(*

.. <legal notes>

legal notes
=================
| SPDX-FileCopyrightText: © 2026 Oleksandr Tiutyk <trofimich@gmail.com>
| SPDX-License-Identifier: LGPL-3.0-only
| For details check: LGPL-3.0-only_

.. _LGPL-3.0-only: https://www.gnu.org/licenses/lgpl-3.0.en.html

.. </legal notes>

*)

FUNCTION_BLOCK ABSTRACT AutomationController 
VAR_GENERIC CONSTANT
    _DeviceCount : INT(0..1000) := 0;
END_VAR
EXTENDS Automation.AutomationComponent IMPLEMENTS IAutomationController
VAR
	_ExceptionHandler : Core.IExceptionHandler;

	_State : AUTOMATION_CONTROLLER_STATE;	
	_PreviousState : AUTOMATION_CONTROLLER_STATE;	

	_Diagnostics : AUTOMATION_CONTROLLER_DIAGNOSTICS;
END_VAR

{attribute 'monitoring' := 'call'}
PROPERTY DeviceCount : INT
GET
DeviceCount := _DeviceCount;
END_GET
END_PROPERTY

{attribute 'monitoring' := 'call'}
PROPERTY ABSTRACT Devices : REFERENCE TO ARRAY [0.._DeviceCount - 1] OF Automation.IDevice
GET
END_GET
END_PROPERTY

{attribute 'monitoring' := 'call'}
PROPERTY FINAL Diagnostics : REFERENCE TO AUTOMATION_CONTROLLER_DIAGNOSTICS
GET
Diagnostics REF= _Diagnostics;
END_GET
END_PROPERTY

METHOD FINAL Disable
VAR
	i : INT;

	exceptionCode : __SYSTEM.ExceptionCode;
	exception : Core.IException;
END_VAR
__TRY
	IF _Enabled THEN
		OnEnabledChanging(FALSE);
	END_IF
	
	IF __ISVALIDREF(Devices) AND_THEN _DeviceCount > 0 THEN
		FOR i := 0 TO _DeviceCount - 1 DO
			Devices[i].Disable();
		END_FOR	
	END_IF

	IF _Enabled THEN	
		_Enabled := FALSE;
		
		OnEnabledChanged();
	END_IF
__CATCH(exceptionCode)	
	_State := AUTOMATION_CONTROLLER_STATE.FAULT;

	exception := Core.ExceptionManager.GetLastException(exceptionCode);	

	fillErrorLog('LastDisableError', Diagnostics.LastDisableError, exception);					
__ENDTRY
END_METHOD

METHOD FINAL Enable
VAR_INPUT
	includeChildren : BOOL := TRUE;
END_VAR
VAR
	i : INT;

	exceptionCode : __SYSTEM.ExceptionCode;
	exception : Core.IException;
END_VAR
__TRY
	IF NOT _Enabled THEN
		OnEnabledChanging(TRUE);
	END_IF
	
	IF includeChildren AND_THEN __ISVALIDREF(Devices) AND_THEN _DeviceCount > 0 THEN
		FOR i := 0 TO _DeviceCount - 1 DO
			Devices[i].Enable();
		END_FOR	
	END_IF
	
	IF NOT _Enabled THEN
		_Enabled := TRUE;
		
		OnEnabledChanged();
	END_IF
__CATCH(exceptionCode)	
	_State := AUTOMATION_CONTROLLER_STATE.FAULT;

	exception := Core.ExceptionManager.GetLastException(exceptionCode);	

	fillErrorLog('LastEnableError', Diagnostics.LastEnableError, exception);					
__ENDTRY
END_METHOD

PROPERTY FINAL ExceptionHandler : Core.IExceptionHandler
GET
ExceptionHandler := _ExceptionHandler;
END_GET
SET
_ExceptionHandler := ExceptionHandler;
END_SET
END_PROPERTY

METHOD FINAL Execute
VAR
	invalidStateException : Core.StandardException;
END_VAR
_PreviousState := _State;

IF NOT Enabled THEN
	RETURN;
END_IF

IF _State = AUTOMATION_CONTROLLER_STATE.INITIAL THEN
	invalidStateException.Throw(NamespaceName, ClassName, __POUNAME(), __POSITION(), "Automation controller is not initialized");
END_IF

handleInputDevices();

handleWorkingStates();

handleOutputDevices();
END_METHOD

METHOD FB_init : BOOL
VAR_INPUT
	(* if TRUE, the retain variables are initialized (warm start / cold start)*)
	bInitRetains	: BOOL;
	(* if TRUE, the instance afterwards gets moved into the copy code (online change)*)
	bInCopyCode	: BOOL;
	name : WSTRING;
END_VAR
_Name := SEL(Core.WideStrings.IsNullOrWhiteSpace(name), name, GetDefaultName());
END_METHOD

METHOD PRIVATE fillErrorLog
VAR_INPUT
	errorPlace : STRING(39);
END_VAR
VAR_IN_OUT
	targetErrorLog : AUTOMATION_ERROR_LOG;
	sourceException : Core.IException;  
END_VAR
_Diagnostics.LastErrorPalce := errorPlace;

targetErrorLog.ShortMessage := sourceException.GetMessage(FALSE, FALSE);
targetErrorLog.FullMessage := sourceException.GetMessage(TRUE, TRUE);
targetErrorLog.Source := sourceException.GetSourceDescription();
targetErrorLog.LocalTimestamp := sourceException.LocalTimestamp;
targetErrorLog.UtcTimestamp := sourceException.UtcTimestamp;

Core.LogManager.TryLogException(sourceException, "AutomationControllerError");
END_METHOD

METHOD PRIVATE handleInputDevices
VAR
	i : DINT;

	exceptionCode : __SYSTEM.ExceptionCode;
	exception : Core.IException;
	
	inputDevice : Automation.IInputDevice;
END_VAR
IF __ISVALIDREF(Devices) AND_THEN _DeviceCount > 0 THEN
	FOR i := 0 TO _DeviceCount - 1 DO
		IF NOT Devices[i].Enabled OR_ELSE NOT __QUERYINTERFACE(Devices[i], inputDevice) THEN
			CONTINUE;
		END_IF
		
		__TRY
			inputDevice.ProcessInput();
		__CATCH(exceptionCode)
			exception := Core.ExceptionManager.GetLastException(exceptionCode);
						
			fillErrorLog('LastRefreshInputDeviceError', Diagnostics.LastRefreshInputDeviceError, exception);
					
			IF _State <> AUTOMATION_CONTROLLER_STATE.FAULT THEN
				setState(AUTOMATION_CONTROLLER_STATE.FAULT);				
			END_IF					
		__ENDTRY
	END_FOR
END_IF
END_METHOD

METHOD PRIVATE handleOutputDevices
VAR
	i : DINT;

	exceptionCode : __SYSTEM.ExceptionCode;
	exception : Core.IException;
	
	outputDevice : Automation.IOutputDevice;	
END_VAR
IF __ISVALIDREF(Devices) AND_THEN _DeviceCount > 0 THEN
	FOR i := 0 TO _DeviceCount - 1 DO
		IF NOT Devices[i].Enabled OR_ELSE NOT __QUERYINTERFACE(Devices[i], outputDevice) THEN
			CONTINUE;
		END_IF
		
		__TRY
			outputDevice.ProcessOutput(); 
		__CATCH(exceptionCode)
			exception := Core.ExceptionManager.GetLastException(exceptionCode);
						
			fillErrorLog('LastRefreshOutputDeviceError', Diagnostics.LastRefreshOutputDeviceError, exception);

			IF _State <> AUTOMATION_CONTROLLER_STATE.FAULT THEN
				setState(AUTOMATION_CONTROLLER_STATE.FAULT);				
			END_IF					
		__ENDTRY 
	END_FOR
END_IF
END_METHOD

METHOD PRIVATE handleWorkingStates
VAR
	i : DINT;

	exceptionCode : __SYSTEM.ExceptionCode;
	exception : Core.IException;
END_VAR
__TRY
	CASE _State OF
		AUTOMATION_CONTROLLER_STATE.WORKING:
			OnWorking();
			
		AUTOMATION_CONTROLLER_STATE.FAULT:
			OnFault();
			
		AUTOMATION_CONTROLLER_STATE.RESETTING:			
			IF OnResetting() THEN
				setState(AUTOMATION_CONTROLLER_STATE.WORKING);
			END_IF			
	END_CASE
__CATCH(exceptionCode)	
	exception := Core.ExceptionManager.GetLastException(exceptionCode);	

	CASE _State OF
		AUTOMATION_CONTROLLER_STATE.WORKING:
			fillErrorLog('LastRunningError', Diagnostics.LastRunningError, exception);			

		AUTOMATION_CONTROLLER_STATE.FAULT:
			fillErrorLog('LastFaultError', Diagnostics.LastFaultError, exception);
					
		AUTOMATION_CONTROLLER_STATE.RESETTING:		
			fillErrorLog('LastResettingError', Diagnostics.LastResettingError, exception);					
	END_CASE
	
	IF _ExceptionHandler = 0 OR_ELSE NOT _ExceptionHandler.HandleException(exception) THEN
		setState(AUTOMATION_CONTROLLER_STATE.FAULT);
	END_IF						
__ENDTRY
END_METHOD

METHOD FINAL Initialize : BOOL
VAR
	i : DINT;

	exceptionCode : __SYSTEM.ExceptionCode;
	exception : Core.IException;
	
	deviceNotSpecifiedException : Core.DataMemberNotSpecifiedException;
END_VAR
IF _State <> AUTOMATION_CONTROLLER_STATE.INITIAL THEN
	RETURN;
END_IF

__TRY
	IF _DeviceCount > 0 AND_THEN NOT __ISVALIDREF(Devices) THEN
		deviceNotSpecifiedException.Throw(Namespacename, ClassName, __POUNAME(), __POSITION(), 'Devices');
	END_IF
	
	OnPreDeviceInitializing();
	
	Initialize := TRUE;

	IF _DeviceCount > 0 THEN
		FOR i := 0 TO _DeviceCount - 1 DO
			IF Devices[i] = 0 THEN
				deviceNotSpecifiedException.Throw(Namespacename, ClassName, __POUNAME(), __POSITION(), Core.Strings.Concat255('Devices[', TO_STRING(i), ']'));			
			END_IF
			
			Initialize := Initialize AND Devices[i].Initialize();
		END_FOR
	END_IF

	Initialize := Initialize AND OnPostDeviceInitializing();
	
	IF Initialize THEN
		setState(AUTOMATION_CONTROLLER_STATE.WORKING);
	END_IF	
__CATCH(exceptionCode)
	setState(AUTOMATION_CONTROLLER_STATE.FAULT);
	
	exception := Core.ExceptionManager.GetLastException(exceptionCode);
					
	fillErrorLog('InitializationError', Diagnostics.InitializationError, exception);					
__ENDTRY
END_METHOD

METHOD PROTECTED OnEnabledChanged
END_METHOD

METHOD PROTECTED OnEnabledChanging
VAR_INPUT
	newValue : BOOL;
END_VAR
END_METHOD

METHOD PROTECTED OnFault
END_METHOD

METHOD PROTECTED OnPostDeviceInitializing : BOOL
OnPostDeviceInitializing := TRUE;
END_METHOD

METHOD PROTECTED OnPreDeviceInitializing
END_METHOD

METHOD PROTECTED OnResetting : BOOL
OnResetting := TRUE;
END_METHOD

METHOD PROTECTED ABSTRACT OnWorking
END_METHOD

METHOD FINAL Reset : BOOL
VAR_OUTPUT
	refuseReason : WSTRING(255);
END_VAR
IF _State <> AUTOMATION_CONTROLLER_STATE.FAULT THEN
	refuseReason := Core.WideStrings.Concat255("Expected controller state is 'FAULT', but actual controller state is '", TO_WSTRING(_State), "'");
	RETURN;
END_IF

setState(AUTOMATION_CONTROLLER_STATE.RESETTING);

Reset := TRUE;
END_METHOD

METHOD PRIVATE setState
VAR_INPUT
	state : AUTOMATION_CONTROLLER_STATE;
END_VAR
_PreviousState := _State;
_State := state;
END_METHOD

{attribute 'monitoring' := 'call'}
PROPERTY FINAL State : AUTOMATION_CONTROLLER_STATE
GET
State := _State;
END_GET
END_PROPERTY

{attribute 'monitoring' := 'call'}
PROPERTY FINAL StateChanged : BOOL
GET
StateChanged := _State <> _PreviousState;
END_GET
END_PROPERTY

{attribute 'monitoring' := 'call'}
PROPERTY StateName : STRING
GET
StateName := TO_STRING(_State);
END_GET
END_PROPERTY

METHOD FINAL TryGetDeviceByIndex : Automation.IDevice
VAR_INPUT
	index : BYTE;
END_VAR
IF index < 0 OR_ELSE index >= _DeviceCount OR_ELSE NOT __ISVALIDREF(Devices) THEN
	RETURN;
END_IF

TryGetDeviceByIndex := Devices[index];
END_METHOD

END_FUNCTION_BLOCK

(* stored: Version 1.1.0.1
   POU AutomationController: Id {715bcab9-6d21-43bf-ac33-fb2affdac1da}, SpecialFunc None
   Folder Methods to override: Id {18713aca-9c47-4769-936e-cd3be2ed069c}
   Folder EnabledChange: Id {7cc34a9f-6118-4793-9de6-359b78cb7be4}
   Folder Initialization: Id {42d1bd21-062f-45b1-a165-3fc00e8443d8}
   Folder Service memebers: Id {5df4ad11-a7ac-4049-8c04-41c0497c7559}
   Property DeviceCount: Id {612962ce-4a03-4dcb-a1ce-f9e94eefa0eb}
   Get Get: Id {cc518b3a-e440-4848-8075-189e5ee4e093}
   Property Devices: Id {f1c94009-408f-4558-836f-c0ffe07e995d}
   Get Get: Id {3053aa14-2407-42d1-bc4d-bd38e5a9f72c}
   Property Diagnostics: Id {89d80bd2-f2bc-45f4-b861-f9194e4bb6a5}
   Get Get: Id {6974a2c5-c336-4c3a-a18a-82f762fc3656}
   Method Disable: Id {94567983-f3f5-4266-9cfb-3c5f4ea14259}
   Method Enable: Id {df8c9490-4eb4-4f45-9a7b-8c348978a15b}
   Property ExceptionHandler: Id {60a29608-799c-49a7-a0f5-81ee4e55824c}
   Get Get: Id {fae050a0-52d3-4847-a89b-06de749e48ee}
   Set Set: Id {0ab07e6b-d588-44a7-8de9-0695649fe2c2}
   Method Execute: Id {edf960fe-6c94-4ace-a7be-524e71aafd2a}
   Method FB_init: Id {9b3a4632-16b8-4d26-a6b5-e8140364c2cb}
   Method fillErrorLog: Id {13ecfb4e-9729-40c0-b5b7-a5c89543cb1f}
   Method handleInputDevices: Id {cd23818a-f724-4bce-970a-f4c5c7f1d1fb}
   Method handleOutputDevices: Id {421f0782-6afa-4e82-84cb-a5cc3ea35f21}
   Method handleWorkingStates: Id {bb165360-ba12-474f-a548-167a2e5dd0a1}
   Method Initialize: Id {eb1221b0-f976-4a46-99f2-a6494cff3a27}
   Method OnEnabledChanged: Id {dd63764b-f122-4f50-a25d-0df5144930d7}
   Method OnEnabledChanging: Id {d1fcb6d0-b53a-4b1a-b954-eb5cd2d33bc4}
   Method OnFault: Id {47b787a0-74db-428e-a805-17453cf9f9ee}
   Method OnPostDeviceInitializing: Id {b196f5d6-1614-4d95-80dc-69c224e94b14}
   Method OnPreDeviceInitializing: Id {f30a4c4a-7966-446f-95b6-a1ce70efb536}
   Method OnResetting: Id {26bb7324-2a54-4dd6-91d7-07c8f2cb1be0}
   Method OnWorking: Id {ebc39867-3255-43ca-899d-74387b198a9b}
   Method Reset: Id {d15376e1-1a99-49f6-b2b0-b5cf3e7f7e51}
   Method setState: Id {9b9897ff-6da5-467a-bc24-ba7a46c549d1}
   Property State: Id {b57e32a3-ebf4-4492-89c3-02193601134f}
   Get Get: Id {e675c2b5-5934-4e03-a0b0-61bb8b8e344b}
   Property StateChanged: Id {2d2d514b-9477-4fbb-b4e8-52562c635954}
   Get Get: Id {c4932c37-19e2-4343-9ad0-6d106776d675}
   Property StateName: Id {1f460bbf-201a-476c-9987-4ccb4784c5c5}
   Get Get: Id {4fed4a37-5097-4a72-961f-12fff28b9f42}
   Method TryGetDeviceByIndex: Id {822b2535-548b-4af3-814e-271dc3e4c03f} *)
